// TwinCAT 3 PLC project PlcSoftware
// ProgramVersion: 3.1.4022.7
// libraries:
//   AST_V1_0, * (Deprag)
//   Tc2_MC2, * (Beckhoff Automation GmbH)
//   Tc2_MC2_Drive, * (Beckhoff Automation GmbH)
//   Tc2_Standard, * (Beckhoff Automation GmbH)
//   Tc2_System, * (Beckhoff Automation GmbH)
//   Tc2_Utilities, * (Beckhoff Automation GmbH)
//   Tc3_Module, * (Beckhoff Automation GmbH)
//   Tc3_PLCopen_OpcUa, * (Beckhoff Automation GmbH)
// project tree:
//   DUTs/ENUMs/ teAxisNames.TcDUT, teDriveState.TcDUT, teOperationMode.TcDUT, teScrewFeeders.TcDUT
//   DUTs/STRUCTs/ tsASTData.TcDUT, tsAxisPositionPoint.TcDUT, tsAxisPositions.TcDUT (not stored), tsControls.TcDUT, tsCoordinate.TcDUT, tsCoordinateBool.TcDUT (not stored), tsDriveOutputs.TcDUT, tsDriveParameter.TcDUT, tsRecipe.TcDUT (not stored), tsRecipeRow.TcDUT (not stored)
//   FBs/DRIVEs/AXIS/ FB_PTP_AXIS_ABS_CONTROL.TcPOU
//   FBs/DRIVEs/PNEU/ PNEU_DRIVE.TcPOU
//   FBs/RECIPEs/CONVERTERs/ ConvertCommandToString.TcPOU, CovertStringToCommand.TcPOU
//   FBs/RECIPEs/FILEs/ CreateRecipeFile.TcPOU, ReadRecipeFromFile.TcPOU, WriteRepcieToFile.TcPOU
//   FBs/SUBFUNCTIONs/ BLOW_DOW_SEQ.TcPOU, END_RUN_SEQ.TcPOU, HOME_RUN_SEQ.TcPOU, PICKUP_SCREW_SEQ.TcPOU, SELECT_ACTIVE_FEEDER_SEQ.TcPOU
//   GVLs/ AST40_GLV.TcGVL, CTRL_GVL.TcGVL, HMI_GLV.TcGVL, IN_OUT_GLV.TcGVL, PERSIST_GLV.TcGVL, SAFETY_IN_GLV.TcGVL, SAFETY_OUT_GLV.TcGVL
//   POUs/JIG POUs/JIG TYPE POUs/ JIG_EMPTY.TcPOU, JIG_GRAB.TcPOU, JIG_PARTPRESENT.TcPOU, JIG_TAKER.TcPOU
//   POUs/JIG POUs/ JIG001_VOLVOL125.TcPOU, JIG002_MANSCANIA2016.TcPOU, JIG003_NTG6.TcPOU, JIG004_BMW_RAM.TcPOU, JIG005_BMW_MGU.TcPOU
//   POUs/KERNEL POUs/ AST40_Controller.TcPOU, HMI_Controller.TcPOU, INIT_DataSet.TcPOU, MES_Controller.TcPOU, MOVMENT_Controller.TcPOU, OPERATION_Controller.TcPOU, RECIPE_Controller.TcPOU
//   POUs/KERNEL POUs/MES POUs/ LOCAL_COM_Controller.TcPOU, OPCUA_Controller.TcPOU
//   POUs/KERNEL POUs/OPERATIONs/ AUTOMATIC_POSITION_TEST.TcPOU, AUTOMATIC_SCREWING.TcPOU, AUTOMATIC_SCREW_PICKUP_TEST.TcPOU
//   POUs/KERNEL POUs/OPERATIONs/SUBOPERATIONs/ DROP_SCREW.TcPOU, END_RUN.TcPOU, HOME_RUN.TcPOU, PICKUP_SCREW.TcPOU, POSITION_RUN.TcPOU
//   POUs/MAIN POUs/ FAST.TcPOU, INDEP.TcPOU, JIG.TcPOU, MAIN.TcPOU
//   TASKs/ FastTask.TcTTO, PlcTask.TcTTO
// real-time tasks:
//   TASK PlcTask: cycle T#10ms, priority 12, ADS port 350
//   TASK FastTask: cycle T#10ms, priority 8, ADS port 351
// motion (NC):
//   TASK NC/PTP Task SAF: cycle T#2ms, priority 4, ADS port 501
//   TASK NC/PTP Task SVB: cycle T#10ms, priority 10, ADS port 511
//   AXIS X Axis (id 5)
//     OtherSettings: AllowMotionCmdToSlave=true
//     encoder EncType=1
//     drive DrvType=5
//       Analog: ScaleFactorActTorque=0.1
//       TimeComp: TaskDelayCycles=1
//     controller CtrType=1
//       CtrPara: PriorControlFactor=1
//         Observer: BandWidth=20
//   AXIS Y Axis (id 6)
//     OtherSettings: AllowMotionCmdToSlave=true
//     encoder EncType=1
//     drive DrvType=5
//       Analog: ScaleFactorActTorque=0.1
//       TimeComp: TaskDelayCycles=1
//     controller CtrType=1
//       CtrPara: PriorControlFactor=1
//         Observer: BandWidth=20
//   AXIS Z Axis (id 7)
//     OtherSettings: AllowMotionCmdToSlave=true
//     encoder EncType=1
//     drive DrvType=5
//       Analog: ScaleFactorActTorque=0.1
//       TimeComp: TaskDelayCycles=1
//     controller CtrType=1
//       CtrPara: PriorControlFactor=1
//         Observer: BandWidth=20
//   AXIS C Axis (id 8)
//     OtherSettings: AllowMotionCmdToSlave=true
//     encoder EncType=1
//     drive DrvType=5
//       Analog: ScaleFactorActTorque=0.1
//       TimeComp: TaskDelayCycles=1
//     controller CtrType=1
//       CtrPara: PriorControlFactor=1
//         Observer: BandWidth=20
//   AXIS Sim X Axis (id 1)
//     OtherSettings: AllowMotionCmdToSlave=true
//     encoder EncType=1
//       SoftEndMinControl: Enable=true, Range=-40
//       SoftEndMaxControl: Enable=true, Range=640
//     drive DrvType=5
//       Analog: ScaleFactorActTorque=0.1
//       TimeComp: TaskDelayCycles=1
//     controller CtrType=1
//       CtrPara: PriorControlFactor=1
//         Observer: BandWidth=20
//   AXIS Sim Y Axis (id 2)
//     OtherSettings: AllowMotionCmdToSlave=true
//     encoder EncType=1
//       SoftEndMinControl: Enable=true, Range=-193
//       SoftEndMaxControl: Enable=true, Range=530
//     drive DrvType=5
//       Analog: ScaleFactorActTorque=0.1
//       TimeComp: TaskDelayCycles=1
//     controller CtrType=1
//       CtrPara: PriorControlFactor=1
//         Observer: BandWidth=20
//   AXIS Sim Z Axis (id 3)
//     OtherSettings: AllowMotionCmdToSlave=true
//     encoder EncType=1
//       SoftEndMinControl: Enable=true, Range=-3
//       SoftEndMaxControl: Enable=true, Range=252
//     drive DrvType=5
//       Analog: ScaleFactorActTorque=0.1
//       TimeComp: TaskDelayCycles=1
//     controller CtrType=1
//       CtrPara: PriorControlFactor=1
//         Observer: BandWidth=20
//   AXIS Sim C Axis (id 4)
//     OtherSettings: AllowMotionCmdToSlave=true
//     encoder EncType=1
//       SoftEndMinControl: Enable=true
//       SoftEndMaxControl: Enable=true
//     drive DrvType=5
//       Analog: ScaleFactorActTorque=0.1
//       TimeComp: TaskDelayCycles=1
//     controller CtrType=1
//       CtrPara: PriorControlFactor=1
//         Observer: BandWidth=20
// variable links:
//   PlcSoftware/PlcSoftware Instance <-> NC/PTP Task SAF/Axes/Sim C Axis
//     PlcTask Inputs/IN_OUT_GLV.G_aAxisReferencies[4].NcToPlc <-> Outputs/ToPlc
//     PlcTask Outputs/IN_OUT_GLV.G_aAxisReferencies[4].PlcToNc <-> Inputs/FromPlc
//   PlcSoftware/PlcSoftware Instance <-> NC/PTP Task SAF/Axes/Sim X Axis
//     PlcTask Inputs/IN_OUT_GLV.G_aAxisReferencies[1].NcToPlc <-> Outputs/ToPlc
//     PlcTask Outputs/IN_OUT_GLV.G_aAxisReferencies[1].PlcToNc <-> Inputs/FromPlc
//   PlcSoftware/PlcSoftware Instance <-> NC/PTP Task SAF/Axes/Sim Y Axis
//     PlcTask Inputs/IN_OUT_GLV.G_aAxisReferencies[2].NcToPlc <-> Outputs/ToPlc
//     PlcTask Outputs/IN_OUT_GLV.G_aAxisReferencies[2].PlcToNc <-> Inputs/FromPlc
//   PlcSoftware/PlcSoftware Instance <-> NC/PTP Task SAF/Axes/Sim Z Axis
//     PlcTask Inputs/IN_OUT_GLV.G_aAxisReferencies[3].NcToPlc <-> Outputs/ToPlc
//     PlcTask Outputs/IN_OUT_GLV.G_aAxisReferencies[3].PlcToNc <-> Inputs/FromPlc

CONFIGURATION PlcSoftware
    RESOURCE PLC ON TwinCAT3
        TASK FastTask(INTERVAL := T#10ms, PRIORITY := 8);
        TASK PlcTask(INTERVAL := T#10ms, PRIORITY := 12);
        PROGRAM FAST WITH FastTask : FAST;
        PROGRAM MAIN WITH PlcTask : MAIN;
    END_RESOURCE
END_CONFIGURATION

// ---- DUTs/ENUMs/teAxisNames.TcDUT
TYPE teAxisNames :
(
	CE_AXIS_X:=1,			// X-axis drive
	CE_AXIS_Y,				// Y-axis drive
	CE_AXIS_Z,				// Z-axis drive
	CE_AXIS_C 				// C-axis drive
);
END_TYPE

// ---- DUTs/ENUMs/teDriveState.TcDUT
TYPE teDriveState :
(
	MOVESTATE_INIT,
	MOVESTATE_ENABLE,
	MOVESTATE_AUTO,
	MOVESTATE_MANUAL,
	MOVESTATE_IDLE,
	MOVESTATE_ERROR,
	MOVESTATE_RESET
) UDINT;
END_TYPE

// ---- DUTs/ENUMs/teOperationMode.TcDUT
TYPE teOperationMode :
(
	OPMODE_REFERENCETEACH,
	OPMODE_AUTOSCREWING,
	OPMODE_PICKUPTEST,
	OPMODE_POSITIONTEST
) UDINT;
END_TYPE

// ---- DUTs/ENUMs/teScrewFeeders.TcDUT
TYPE teScrewFeeders :
(
	CE_SCREW_FEED_1:=1,
	CE_SCREW_FEED_2,
	CE_SCREW_FEED_3,
	CE_SCREW_FEED_4
);
END_TYPE

// ---- DUTs/STRUCTs/tsASTData.TcDUT
TYPE tsASTData :
STRUCT
	Start:			BOOL;
	Prog:			INT;
	DataSaved:		BOOL;
	
	OK:				BOOL;
	NOK:			BOOL;
	Ready:			BOOL;
	DataAvailable:	BOOL;
	
	Status:			INT;
	Step:			DINT;
	MinTorque:		REAL;
	MaxTorque:		REAL;
	Torque:			REAL;
	MinAngle:		DINT;
	MaxAngle:		DINT;
	Angle:			REAL;
	Started:		BOOL;
END_STRUCT
END_TYPE

// ---- DUTs/STRUCTs/tsAxisPositionPoint.TcDUT
TYPE tsAxisPositionPoint :
STRUCT
	Name			: STRING;
	Description		: STRING;
	Target			: LREAL;
END_STRUCT
END_TYPE

// ---- DUTs/STRUCTs/tsControls.TcDUT
TYPE tsControls :
STRUCT
	PowerOn:					BOOL:=TRUE;
	AutoMode:					BOOL:=0;						//Automaic/Manual mode switch
	ErrorExist:					BOOL;  							//Error exist
	ErrorACK:					BOOL;							//Error acknowledge
	ManualMoveMode:				BOOL:=TRUE;						//0:= stepper, 1:= continous
	
	OperationMode:				INT:=1;							//0:= manual, 1:= automatic seq 01 ... 

	Override:					LREAL:=100;						//Main overrride value
	ManualOverride:				LREAL:=20;						//Maximum manual override value
	StepSize:					LREAL:=0.1;						//Manual jog step size
	MaximumVelocity:			LREAL:=600;						//Maximum velocity
	
	ActualPosition:				tsCoordinate;	
	TargetPosition:				tsCoordinate;	
END_STRUCT
END_TYPE

// ---- DUTs/STRUCTs/tsCoordinate.TcDUT
TYPE tsCoordinate :
STRUCT
	X: LREAL;
	Y: LREAL;
	Z: LREAL;
	C: LREAL;
END_STRUCT
END_TYPE

// ---- DUTs/STRUCTs/tsDriveOutputs.TcDUT
TYPE tsDriveOutputs :
STRUCT
	PowerOut: 			ST_McOutputs;
	ResetOut: 				ST_McOutputs;
	MoveAbsoluteOut: 		ST_McOutputs;
	MoveJogOut:				ST_McOutputs;
	MoveHalt:				ST_McOutputs;
END_STRUCT
END_TYPE

// ---- DUTs/STRUCTs/tsDriveParameter.TcDUT
TYPE tsDriveParameter :
STRUCT
	PositionMin:		LREAL;
	PositionMax:		LREAL;
	PositionOffset:		LREAL;	
END_STRUCT
END_TYPE

// ---- GVLs/AST40_GLV.TcGVL
VAR_GLOBAL
	G_sAST40_Data:				tsASTData;					//Contains all of AST40 datas	
	
	G_fbAST40:				FB_AST40;					// FB instance of the AST40
	G_sAST40:				tAST40;						// struct contains 'control', 'state' and 'data'
	
	G_sTx					AT%I*: tAST40Rx; 			// struct for the input mapping 
	G_sRx 					AT%Q*: tAST40Tx; 			// struct for the output mapping
END_VAR

// ---- GVLs/CTRL_GVL.TcGVL
VAR_GLOBAL
	G_sControl:						tsControls;						//Control data	

	G_sAxisReady:					tsCoordinateBool;				//Axis ready to move state container
	G_sAxisDone:					tsCoordinateBool;				//Axis done state container
	G_sAckAxisDone:					tsCoordinateBool;				//Axis done acknowledge container
	
	G_sStartToPos:					tsCoordinateBool;				//Start to position
END_VAR

// ---- GVLs/HMI_GLV.TcGVL
VAR_GLOBAL
	G_sHMIAxisJogForward:				tsCoordinateBool;				//Axis jog forward
	G_sHMIAxisJogBackward:				tsCoordinateBool;				//Axis jog backward
END_VAR

// ---- GVLs/IN_OUT_GLV.TcGVL
VAR_GLOBAL
	//Axis referencies for driving
	G_aAxisReferencies:				ARRAY [1..CE_AXIS_C] OF AXIS_REF;
	
	//Input linkable definition
	I_xFeedbackES           		AT%I* :BOOL;
	I_xVacuumIntake_OK				AT%I*: BOOL;
	I_xStart						AT%I*: BOOL;
	I_xLightGridError				AT%I*: BOOL;
	I_xSafetyDoorClosed				AT%I*: BOOL;
	I_xServoFanDiag					AT%I*: BOOL;
	I_xPneumatic_OK					AT%I*: BOOL;
	I_xScrewFeed_READY			 	AT%I*: ARRAY[1..CE_SCREW_FEED_4] OF BOOL;
	I_xScrewFeeder_POS				AT%I*: ARRAY[1..CE_SCREW_FEED_4] OF BOOL;
	I_xPartSensor1					AT%I*: BOOL;
	I_xPartSensor2					AT%I*: BOOL;
	I_xEpInputBox01					AT%I*: ARRAY[1..16] OF BOOL;	
	I_xEpInputBox02					AT%I*: ARRAY[1..16] OF BOOL;
	
	//Output linkable definition
	Q_axScrewFeeders					AT%Q*:ARRAY [1..CE_SCREW_FEED_4] OF BOOL;
	Q_xValve_PressureSwitch				AT%Q*: BOOL;
	Q_xBlowValve						AT%Q*: BOOL;
	Q_xVacuumValve						AT%Q*: BOOL;
END_VAR

// ---- GVLs/PERSIST_GLV.TcGVL
VAR_GLOBAL PERSISTENT
	G_xExistCAxis:					BOOL:=TRUE;							//TRUE:=Exist C-Axis, FALSE:=Not exist C-Axis
	//Individual axis positions like fider position...
	G_asIndividualAxisPositions:		ARRAY [1..CE_AXIS_C] OF tsAxisPositions;
	//Min/Max/Offset parameters for drives...
	G_asDriveParameters:				ARRAY [1..CE_AXIS_C] OF tsDriveParameter:= [(PositionMin:=-40.00,	PositionMax:=640.00,		PositionOffset:=-293.00),	(*X-Axis initial parameters*)
																					(PositionMin:=-193.00,	PositionMax:=530.00,	PositionOffset:=240.00),		(*Y-Axis initial parameters*)
																					(PositionMin:=-3,		PositionMax:=252,		PositionOffset:=127.00), 		(*Z-Axis initial parameters*)
																					(PositionMin:=0,		PositionMax:=0,			PositionOffset:=0.00)];			(*C-Axis initial parameters*)
END_VAR

// ---- GVLs/SAFETY_IN_GLV.TcGVL
VAR_GLOBAL
	I_xTsEstopCH1					AT%I*: BOOL;
	I_xTsEstopCH2					AT%I*: BOOL;
	I_xTsE_Stop			 			AT%I*: BOOL;
	I_xTsCommErr					AT%I*: BOOL;
	I_xTsLightGridOK				AT%I*: BOOL;
	I_xTsFBErr						AT%I*: BOOL;
END_VAR

// ---- GVLs/SAFETY_OUT_GLV.TcGVL
VAR_GLOBAL
	Q_xTsFB_E_Stop					AT%Q*: BOOL;
	Q_xTsEStopReset                 AT%Q*: BOOL;
	Q_xTsTwinsafeRun				AT%Q*: BOOL;
	Q_xTsErrAck						AT%Q*: BOOL;
END_VAR

// ---- POUs/MAIN POUs/FAST.TcPOU
PROGRAM FAST
VAR
	tpEStopAck:		TP;
	rtErrorACK: 	R_TRIG;
END_VAR


Q_xTsTwinsafeRun := NOT I_xTsCommErr;
Q_xTsErrAck := I_xTsCommErr;

rtErrorAck(CLK:= G_sControl.ErrorAck, Q=> G_sControl.ErrorAck);
tpEStopAck(IN:= rtErrorAck.Q, pt:= T#100MS);

Q_xTsFB_E_Stop :=I_xFeedbackES;
Q_xTsEstopReset := (tpEStopAck.ET > T#100MS AND tpEStopAck.ET < T#300MS);

END_PROGRAM

// ---- POUs/MAIN POUs/MAIN.TcPOU
PROGRAM MAIN
VAR
	bInit:					BOOL:=TRUE;	
	xOpenVisu:				BOOL;
	sMachineName:			STRING;
	sVisuURL:				STRING;
	fbStartProcess:			NT_StartProcess;
	fbGetHostName:			FB_GetHostName;
END_VAR

(*
fbGetHostName(	 
				 bExecute:= TRUE,
				 sHostName=>sMachineName);
sVisuURL:= CONCAT('--app=https://huszwsap10:1020/Default.html?TargetHost=', sMachineName);
fbStartProcess(
				 NETID:= '',
				 PATHSTR:= 'C:\Program Files (x86)\Google\Chrome\Application\chrome.exe',
				 DIRNAME:= 'C:\Program Files (x86)\Google\Chrome\Application',
				 COMNDLINE:= sVisuURL,
				 START:= (LEN (sMachineName)>0),
				 TMOUT:= T#20S);
*)		
		 
INIT_DataSet();
//RECIPE_Controller();
//DRIVE_Controller();
MOVMENT_Controller();
OPERATION_Controller();
HMI_Controller();

END_PROGRAM

// ---- POUs/KERNEL POUs/INIT_DataSet.TcPOU
PROGRAM INIT_DataSet
VAR
	xWriteExecute:					BOOL;
	xErrorInProces:					BOOL:=FALSE;
	xCounter:						INT:=1;
	
	fbMC_WriteOffsetParameterX: 		MC_WriteParameter;
	fbMC_WriteMinParameterX: 		MC_WriteParameter;
	fbMC_WriteMaxParameterX: 		MC_WriteParameter;
	
	fbMC_WriteOffsetParameterY: 		MC_WriteParameter;
	fbMC_WriteMinParameterY: 		MC_WriteParameter;
	fbMC_WriteMaxParameterY: 		MC_WriteParameter;
	
	fbMC_WriteOffsetParameterZ: 		MC_WriteParameter;
	fbMC_WriteMinParameterZ: 		MC_WriteParameter;
	fbMC_WriteMaxParameterZ: 		MC_WriteParameter;
	
	fbMC_WriteOffsetParameterC: 		MC_WriteParameter;
	fbMC_WriteMinParameterC: 		MC_WriteParameter;
	fbMC_WriteMaxParameterC: 		MC_WriteParameter;
END_VAR

//X-Axis Write parameter
fbMC_WriteOffsetParameterX(
					Axis:= G_aAxisReferencies[CE_AXIS_X], 
					Execute:= xWriteExecute, 
					ParameterNumber:= 1042, 
					Value:= G_asDriveParameters[CE_AXIS_X].PositionOffset,
					Error=>  xErrorInProces
					);
fbMC_WriteMinParameterX(
					Axis:= G_aAxisReferencies[CE_AXIS_X], 
					Execute:= xWriteExecute, 
					ParameterNumber:= 3, 
					Value:= G_asDriveParameters[CE_AXIS_X].PositionMin,
					Error=>  xErrorInProces
					);
fbMC_WriteMaxParameterX(
					Axis:= G_aAxisReferencies[CE_AXIS_X], 
					Execute:= xWriteExecute, 
					ParameterNumber:= 2, 
					Value:= G_asDriveParameters[CE_AXIS_X].PositionMax,
					Error=>  xErrorInProces
					);
//Y-Axis Write paramater
fbMC_WriteOffsetParameterY(
					Axis:= G_aAxisReferencies[CE_AXIS_Y], 
					Execute:= xWriteExecute, 
					ParameterNumber:= 1042, 
					Value:= G_asDriveParameters[CE_AXIS_Y].PositionOffset,
					Error=>  xErrorInProces
					);
fbMC_WriteMinParameterY(
					Axis:= G_aAxisReferencies[CE_AXIS_Y], 
					Execute:= xWriteExecute, 
					ParameterNumber:= 3, 
					Value:= G_asDriveParameters[CE_AXIS_Y].PositionMin,
					Error=>  xErrorInProces
					);
fbMC_WriteMaxParameterY(
					Axis:= G_aAxisReferencies[CE_AXIS_Y], 
					Execute:= xWriteExecute, 
					ParameterNumber:= 2, 
					Value:= G_asDriveParameters[CE_AXIS_Y].PositionMax,
					Error=>  xErrorInProces
					);
//Z-Axis Write parameter
fbMC_WriteOffsetParameterZ(
					Axis:= G_aAxisReferencies[CE_AXIS_Z], 
					Execute:= xWriteExecute, 
					ParameterNumber:= 1042, 
					Value:= G_asDriveParameters[CE_AXIS_Z].PositionOffset,
					Error=>  xErrorInProces
					);
fbMC_WriteMinParameterZ(
					Axis:= G_aAxisReferencies[CE_AXIS_Z], 
					Execute:= xWriteExecute, 
					ParameterNumber:= 3, 
					Value:= G_asDriveParameters[CE_AXIS_Z].PositionMin,
					Error=>  xErrorInProces
					);
fbMC_WriteMaxParameterZ(
					Axis:= G_aAxisReferencies[CE_AXIS_Z], 
					Execute:= xWriteExecute, 
					ParameterNumber:= 2, 
					Value:= G_asDriveParameters[CE_AXIS_Z].PositionMax,
					Error=>  xErrorInProces
					);
//C-Axis Write parameter
fbMC_WriteOffsetParameterC(
					Axis:= G_aAxisReferencies[CE_AXIS_C], 
					Execute:= xWriteExecute, 
					ParameterNumber:= 1042, 
					Value:= G_asDriveParameters[CE_AXIS_C].PositionOffset,
					Error=>  xErrorInProces
					);
fbMC_WriteMinParameterC(
					Axis:= G_aAxisReferencies[CE_AXIS_C], 
					Execute:= xWriteExecute, 
					ParameterNumber:= 3, 
					Value:= G_asDriveParameters[CE_AXIS_C].PositionMin,
					Error=>  xErrorInProces
					);
fbMC_WriteMaxParameterC(
					Axis:= G_aAxisReferencies[CE_AXIS_C], 
					Execute:= xWriteExecute, 
					ParameterNumber:= 2, 
					Value:= G_asDriveParameters[CE_AXIS_C].PositionMax,
					Error=>  xErrorInProces
					);
					
IF xErrorInProces THEN
	xWriteExecute:= FALSE;
ELSE
	xWriteExecute:= TRUE;
END_IF

END_PROGRAM

// ---- POUs/KERNEL POUs/MOVMENT_Controller.TcPOU
PROGRAM MOVMENT_Controller
VAR
	X_Axis:				FB_PTP_AXIS_ABS_CONTROL;
	Y_Axis:				FB_PTP_AXIS_ABS_CONTROL;
	Z_Axis:				FB_PTP_AXIS_ABS_CONTROL;
	
	eJogMode: 				E_JogMode;
END_VAR

IF (G_sControl.ManualMoveMode) THEN
	eJogMode:= MC_JOGMODE_CONTINOUS;
ELSE
	eJogMode:= MC_JOGMODE_INCHING;
END_IF

ACT_AXIS_CTRL();

ACTION ACT_AXIS_CTRL:
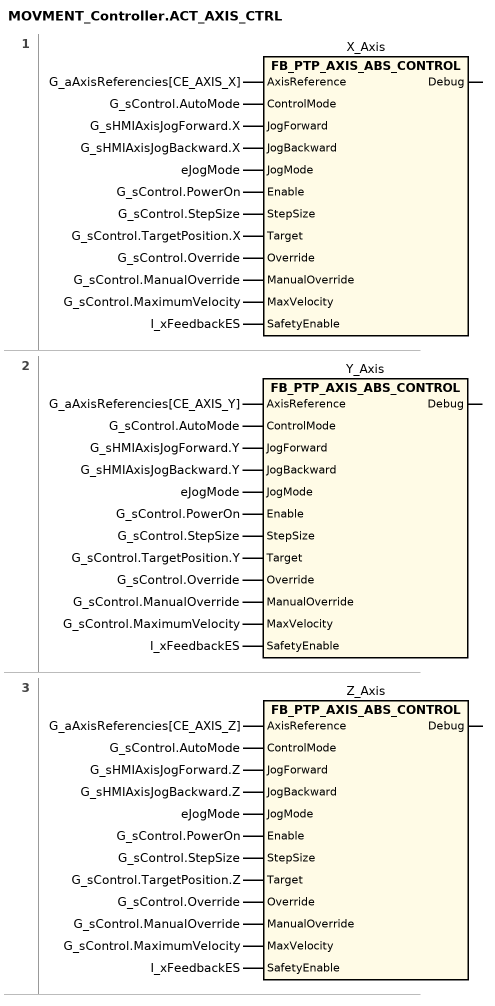
// NETWORK 1
X_Axis(
    AxisReference := G_aAxisReferencies[CE_AXIS_X],
    ControlMode := G_sControl.AutoMode,
    JogForward := G_sHMIAxisJogForward.X,
    JogBackward := G_sHMIAxisJogBackward.X,
    JogMode := eJogMode,
    Enable := G_sControl.PowerOn,
    StepSize := G_sControl.StepSize,
    Target := G_sControl.TargetPosition.X,
    Override := G_sControl.Override,
    ManualOverride := G_sControl.ManualOverride,
    MaxVelocity := G_sControl.MaximumVelocity,
    SafetyEnable := I_xFeedbackES); // FB_PTP_AXIS_ABS_CONTROL

// NETWORK 2
Y_Axis(
    AxisReference := G_aAxisReferencies[CE_AXIS_Y],
    ControlMode := G_sControl.AutoMode,
    JogForward := G_sHMIAxisJogForward.Y,
    JogBackward := G_sHMIAxisJogBackward.Y,
    JogMode := eJogMode,
    Enable := G_sControl.PowerOn,
    StepSize := G_sControl.StepSize,
    Target := G_sControl.TargetPosition.Y,
    Override := G_sControl.Override,
    ManualOverride := G_sControl.ManualOverride,
    MaxVelocity := G_sControl.MaximumVelocity,
    SafetyEnable := I_xFeedbackES); // FB_PTP_AXIS_ABS_CONTROL

// NETWORK 3
Z_Axis(
    AxisReference := G_aAxisReferencies[CE_AXIS_Z],
    ControlMode := G_sControl.AutoMode,
    JogForward := G_sHMIAxisJogForward.Z,
    JogBackward := G_sHMIAxisJogBackward.Z,
    JogMode := eJogMode,
    Enable := G_sControl.PowerOn,
    StepSize := G_sControl.StepSize,
    Target := G_sControl.TargetPosition.Z,
    Override := G_sControl.Override,
    ManualOverride := G_sControl.ManualOverride,
    MaxVelocity := G_sControl.MaximumVelocity,
    SafetyEnable := I_xFeedbackES); // FB_PTP_AXIS_ABS_CONTROL
END_ACTION

END_PROGRAM

// ---- FBs/DRIVEs/AXIS/FB_PTP_AXIS_ABS_CONTROL.TcPOU
FUNCTION_BLOCK FB_PTP_AXIS_ABS_CONTROL
VAR_INPUT
	ControlMode:				BOOL;					// Manual (JOG mode) or Automatic (ABSOLUTE PTP mode) | 0:=Manual 1:=Automatic
	
	JogForward:					BOOL;					// Jog the axis in forward direction (based on the JogMode)
	JogBackward:				BOOL;					// Jog the axis in forward direction (based on the JogMode)
	JogMode:					E_JogMode;				// Selected Jog mode is determin the manual movement method stepper or continous
	
	Enable:						BOOL;					// Enable axis
	Start:						BOOL;					// Start to position in automatic mode
	StepSize:					LREAL;					// Stepsize (like: 0.1mm, 0.2mm, 0.5mm, 1mm ....)
	Target:						LREAL;					// Target position in automatic mode
	Override:					LREAL;					// Overall axis override (0-100%)
	ManualOverride:				LREAL;					// Manual override (0-20%)
	MaxVelocity:				LREAL;					// Maximum axis velocity (0-600)
	
	SafetyEnable:				BOOL;
END_VAR
VAR_IN_OUT
	AxisReference:				AXIS_REF;				// Contains all referencies for the NC Axis
END_VAR
VAR_OUTPUT
	Debug:						tsDriveOutputs;			// Debug function block output struct
END_VAR
VAR
	AxisState:					teDriveState;			// Contains the control actual state.
	
	LastTarget:					LREAL;
	
	MoveAbs:					MC_MoveAbsolute;		
	MoveJog:					MC_Jog;
	MoveHalt:					MC_Halt;
	Reset:						MC_Reset;
	SoEReset:					FB_SoEReset;
	Power:						MC_Power;
END_VAR

(* update the axis status at the beginning of each cycle *)
AxisReference();

(* axis drive state machine *)
CASE AxisState OF
	
	MOVESTATE_INIT:																		(* initialisation *)
		MoveAbs.Execute :=			FALSE;
		Reset.Execute :=			FALSE;
		AxisState := 				MOVESTATE_ENABLE;
		
		IF NOT SafetyEnable THEN 
			AxisState := MOVESTATE_ERROR;
		END_IF
	
	MOVESTATE_ENABLE:																	(* enabel power *)
		Power.Enable :=				TRUE;
		Power.BufferMode :=			MC_Aborting;
		
		IF Power.Status THEN
			AxisState := MOVESTATE_IDLE;
		ELSIF Power.Error THEN
			Power.Enable :=				FALSE;
			AxisState := MOVESTATE_ERROR;
		END_IF
	
	MOVESTATE_IDLE:																		(* Idle state stay here until the next command *)			
		IF ControlMode AND Start AND SafetyEnable THEN
			AxisState := MOVESTATE_AUTO;
			
		ELSIF NOT ControlMode AND (JogForward OR JogBackward) AND SafetyEnable THEN
			AxisState := MOVESTATE_MANUAL;
			
		ELSIF NOT SafetyEnable THEN 
			Power.Enable :=				FALSE;
			AxisState := MOVESTATE_ERROR;
		
		END_IF
		
	MOVESTATE_AUTO:																		(* automatic movment mode *)
		IF LastTarget=target AND NOT Start THEN
			AxisState := MOVESTATE_IDLE;
		ELSE
			MoveAbs.Position := 	target;
			MoveAbs.Velocity := 	MaxVelocity;
			MoveAbs.BufferMode := 	MC_Aborting;
			MoveAbs.Execute := 		TRUE;
			
			IF MoveAbs.Done AND NOT Start THEN
				MoveAbs.Execute := FALSE;
				AxisState := MOVESTATE_IDLE;
				
			ELSIF MoveAbs.CommandAborted OR MoveAbs.Error THEN
				AxisState := MOVESTATE_ERROR;
			END_IF	
		END_IF
	
	MOVESTATE_MANUAL:																	(* manual movement mode *)
		MoveJog.Position := 	StepSize;
		MoveJog.Mode := 		JogMode;
		MoveJog.Velocity := 	(ManualOverride*MaxVelocity)/100;						(* speed reduction in manual movement mode *)
		
		IF MoveJog.Done AND NOT MoveHalt.Done THEN
			MoveHalt.Execute := 	TRUE;
			MoveHalt.BufferMode := 	MC_Aborting;
			
		ELSIF MoveHalt.Done AND NOT MoveJog.Done THEN
				MoveHalt.Execute := FALSE;
				AxisState := MOVESTATE_IDLE;

		ELSIF MoveJog.CommandAborted OR MoveAbs.Error OR MoveHalt.CommandAborted THEN
				AxisState := MOVESTATE_ERROR;	
		END_IF
	
	MOVESTATE_ERROR:																	(* in error state *)
		IF AxisReference.Status.Error THEN
			AxisState := MOVESTATE_RESET;												(* axis error requires reset *)
			
		ELSE
			AxisState := MOVESTATE_INIT;												(* function block errors don't need a reset *)
			
		END_IF
	
	MOVESTATE_RESET:																	(* reset axis functions *)
		Power.Enable :=				FALSE;		
		SoEReset.Execute := TRUE;
		SoEReset.Timeout := T#10S;
		IF NOT SoEReset.Busy THEN
			SoEReset.Execute := FALSE;
			Reset.Execute := TRUE;
			IF Reset.Done THEN
				AxisState := MOVESTATE_INIT;	
			ELSIF Reset.Error THEN
				AxisState := MOVESTATE_INIT; 												(* can't do anything here *)
			END_IF
		END_IF
	
END_CASE

ACT_MOVE();
ACT_POWER();
ACT_RESET();

ACTION ACT_MOVE:
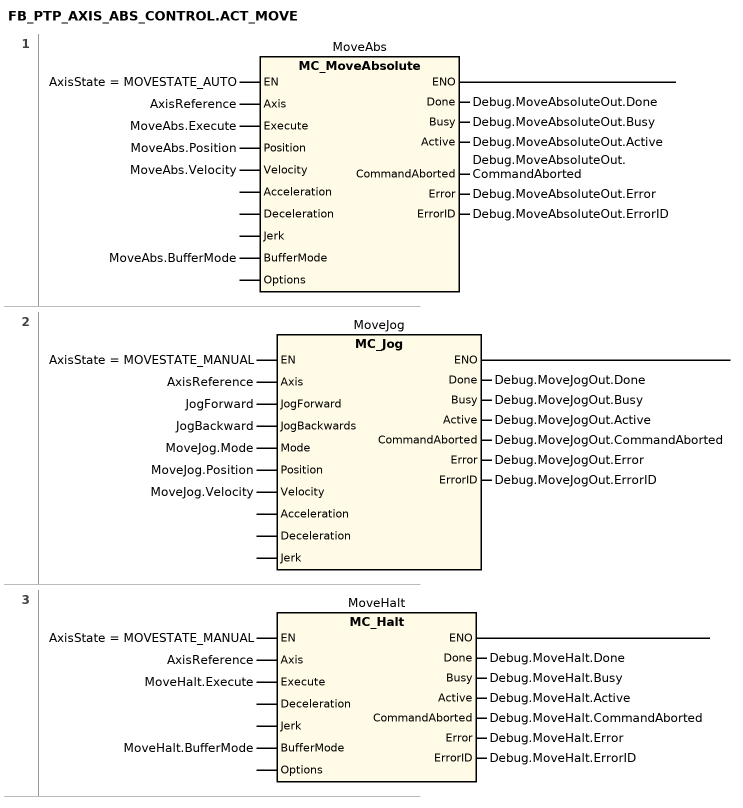
// NETWORK 1
IF AxisState = MOVESTATE_AUTO THEN
    MoveAbs(
        Axis := AxisReference,
        Execute := MoveAbs.Execute,
        Position := MoveAbs.Position,
        Velocity := MoveAbs.Velocity,
        BufferMode := MoveAbs.BufferMode,
        Done => Debug.MoveAbsoluteOut.Done,
        Busy => Debug.MoveAbsoluteOut.Busy,
        Active => Debug.MoveAbsoluteOut.Active,
        CommandAborted => Debug.MoveAbsoluteOut.CommandAborted,
        Error => Debug.MoveAbsoluteOut.Error,
        ErrorID => Debug.MoveAbsoluteOut.ErrorID); // MC_MoveAbsolute
END_IF

// NETWORK 2
IF AxisState = MOVESTATE_MANUAL THEN
    MoveJog(
        Axis := AxisReference,
        JogForward := JogForward,
        JogBackwards := JogBackward,
        Mode := MoveJog.Mode,
        Position := MoveJog.Position,
        Velocity := MoveJog.Velocity,
        Done => Debug.MoveJogOut.Done,
        Busy => Debug.MoveJogOut.Busy,
        Active => Debug.MoveJogOut.Active,
        CommandAborted => Debug.MoveJogOut.CommandAborted,
        Error => Debug.MoveJogOut.Error,
        ErrorID => Debug.MoveJogOut.ErrorID); // MC_Jog
END_IF

// NETWORK 3
IF AxisState = MOVESTATE_MANUAL THEN
    MoveHalt(
        Axis := AxisReference,
        Execute := MoveHalt.Execute,
        BufferMode := MoveHalt.BufferMode,
        Done => Debug.MoveHalt.Done,
        Busy => Debug.MoveHalt.Busy,
        Active => Debug.MoveHalt.Active,
        CommandAborted => Debug.MoveHalt.CommandAborted,
        Error => Debug.MoveHalt.Error,
        ErrorID => Debug.MoveHalt.ErrorID); // MC_Halt
END_IF
END_ACTION

ACTION ACT_POWER:
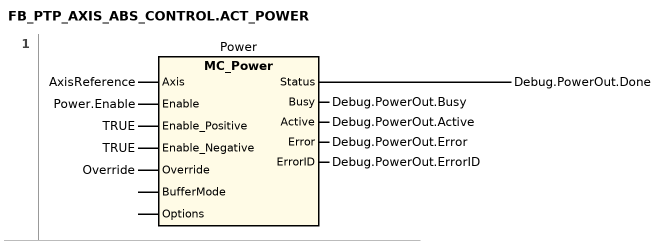
// NETWORK 1
Power(
    Axis := AxisReference,
    Enable := Power.Enable,
    Enable_Positive := TRUE,
    Enable_Negative := TRUE,
    Override := Override,
    Busy => Debug.PowerOut.Busy,
    Active => Debug.PowerOut.Active,
    Error => Debug.PowerOut.Error,
    ErrorID => Debug.PowerOut.ErrorID); // MC_Power
Debug.PowerOut.Done := Power.Status;
END_ACTION

ACTION ACT_RESET:
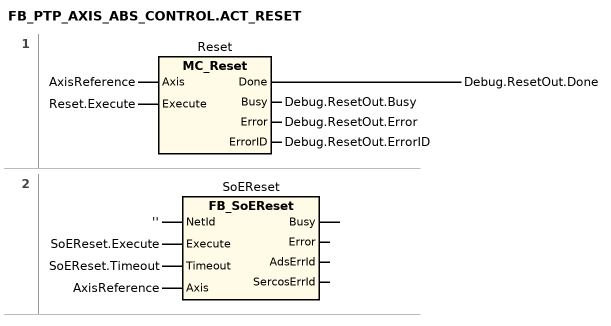
// NETWORK 1
Reset(
    Axis := AxisReference,
    Execute := Reset.Execute,
    Busy => Debug.ResetOut.Busy,
    Error => Debug.ResetOut.Error,
    ErrorID => Debug.ResetOut.ErrorID); // MC_Reset
Debug.ResetOut.Done := Reset.Done;

// NETWORK 2
SoEReset(NetId := '', Execute := SoEReset.Execute, Timeout := SoEReset.Timeout, Axis := AxisReference); // FB_SoEReset
END_ACTION

END_FUNCTION_BLOCK

// ---- POUs/KERNEL POUs/OPERATION_Controller.TcPOU
PROGRAM OPERATION_Controller
VAR	
	xHomeRunExecute:		BOOL;
	xDone:					BOOL;
	xHomeOK:				BOOL;
	
	rtControlOn:			R_TRIG;
	rtHomeRunDone:			R_TRIG;
	
	fbHOME_RUN:				HOME_RUN_SEQ;
END_VAR

rtControlOn(CLK:=G_sControl.AutoMode);
rtHomeRunDone(CLK:=xDone);

IF rtControlOn.Q AND G_sControl.PowerOn AND (NOT G_sControl.ErrorExist) THEN 
	xHomeRunExecute:=TRUE; 
END_IF

IF rtHomeRunDone.Q THEN 
	xHomeOK:=TRUE; 
END_IF

fbHOME_RUN(	xExecute:=xHomeRunExecute, xDone:=xDone);

END_PROGRAM

// ---- FBs/SUBFUNCTIONs/HOME_RUN_SEQ.TcPOU
FUNCTION_BLOCK HOME_RUN_SEQ
VAR_IN_OUT
	xExecute:		BOOL;
	xDone:			BOOL;
END_VAR
VAR_OUTPUT
	
END_VAR
VAR
	tpReset:			TP;
	rtDone:				R_TRIG;
	rtExecute:			R_TRIG;
	ftTimePulse:		F_TRIG;
	tpTimePulse:		TP;
	fbBLOW_DOW_SEQ: 	BLOW_DOW_SEQ;
	xBlowDownExecute:	BOOL;
	fbEND_RUN_SEQ:		END_RUN_SEQ;
	xEndRunExecute:		BOOL;
	
	lrTargetPos:		LREAL;
	xTransCondition:	BOOL;	
	xTransRelease:		BOOL;
	SFCInit:			BOOL;
	SFCReset:			BOOL;	
	SFCError:			BOOL;
	
END_VAR

rtDone(CLK:=xDone);
IF rtDone.Q THEN
	xTransRelease:=FALSE;	
	SFCReset:=TRUE;
	xExecute:=FALSE;
END_IF
rtExecute(CLK:=xExecute);
IF rtExecute.Q THEN
	xTransRelease:=TRUE;
END_IF

aSEQ_ACT();

tpReset(IN:=SFCError, PT:=T#250MS);
SFCReset:= tpReset.Q;

ACTION ACK_DONE_AXIS_active:
IF G_sAxisDone.X OR G_sAxisDone.Y OR G_sAxisDone.Z OR G_sAxisDone.c THEN
	G_sAckAxisDone.X:=TRUE;
	G_sAckAxisDone.Y:=TRUE;
	G_sAckAxisDone.Z:=TRUE;
	G_sAckAxisDone.C:=TRUE;
ELSE
	G_sAckAxisDone.X:=FALSE;
	G_sAckAxisDone.Y:=FALSE;
	G_sAckAxisDone.Z:=FALSE;
	G_sAckAxisDone.C:=FALSE;
END_IF

xTransCondition:= NOT G_sAckAxisDone.X AND NOT G_sAckAxisDone.Y AND NOT G_sAckAxisDone.Z AND NOT G_sAckAxisDone.C;
END_ACTION

ACTION aSEQ_ACT:
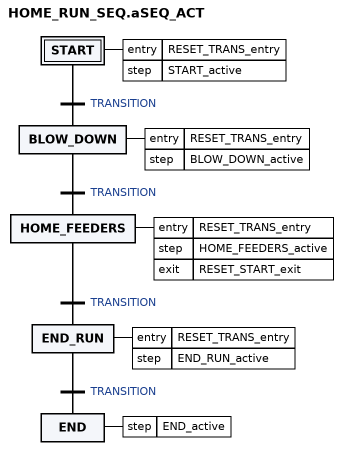
INITIAL_STEP START:
    RESET_TRANS_entry(P1);  // entry action
    START_active(N);  // step action
END_STEP
TRANSITION FROM START TO BLOW_DOWN
    := TRANSITION;
END_TRANSITION
STEP BLOW_DOWN:
    RESET_TRANS_entry(P1);  // entry action
    BLOW_DOWN_active(N);  // step action
END_STEP
TRANSITION FROM BLOW_DOWN TO HOME_FEEDERS
    := TRANSITION;
END_TRANSITION
STEP HOME_FEEDERS:
    RESET_TRANS_entry(P1);  // entry action
    HOME_FEEDERS_active(N);  // step action
    RESET_START_exit(P0);  // exit action
END_STEP
TRANSITION FROM HOME_FEEDERS TO END_RUN
    := TRANSITION;
END_TRANSITION
STEP END_RUN:
    RESET_TRANS_entry(P1);  // entry action
    END_RUN_active(N);  // step action
END_STEP
TRANSITION FROM END_RUN TO END
    := TRANSITION;
END_TRANSITION
STEP END:
    END_active(N);  // step action
END_STEP
END_ACTION

ACTION BLOW_DOWN_active:
xBlowDownExecute:=TRUE;
fbBLOW_DOW_SEQ(	xExecute:=xBlowDownExecute, xDone:=xTransCondition);
END_ACTION

ACTION END_active:
xDone:=TRUE;
xTransCondition:=FALSE;
END_ACTION

ACTION END_RUN_active:
xEndRunExecute:=TRUE;
fbEND_RUN_SEQ(xExecute:=xEndRunExecute,xJigEndDone:=TRUE, xDone:=xTransCondition);
END_ACTION

ACTION HOME_FEEDERS_active:
xTransCondition:=true;
END_ACTION

ACTION RESET_START_exit:
IF G_sAxisDone.X OR G_sAxisDone.Y OR G_sAxisDone.Z OR G_sAxisDone.c THEN
	G_sAckAxisDone.X:=TRUE;
	G_sAckAxisDone.Y:=TRUE;
	G_sAckAxisDone.Z:=TRUE;
	G_sAckAxisDone.C:=TRUE;
ELSE
	G_sAckAxisDone.X:=FALSE;
	G_sAckAxisDone.Y:=FALSE;
	G_sAckAxisDone.Z:=FALSE;
	G_sAckAxisDone.C:=FALSE;
	
	G_sStartToPos.X:=FALSE;
	G_sStartToPos.Y:=FALSE;
	G_sStartToPos.Z:=FALSE;
	G_sStartToPos.C:=FALSE;
END_IF
END_ACTION

ACTION RESET_TRANS_entry:
xTransCondition:= false;
END_ACTION

ACTION START_active:
xDone:=FALSE;
xTransCondition:= NOT xDone;
END_ACTION

TRANSITION TRANSITION:
xTransRelease AND xTransCondition
END_TRANSITION

END_FUNCTION_BLOCK

// ---- FBs/SUBFUNCTIONs/BLOW_DOW_SEQ.TcPOU
FUNCTION_BLOCK BLOW_DOW_SEQ
VAR_IN_OUT
	xExecute:		BOOL;
	xDone:			BOOL;
END_VAR
VAR_OUTPUT
	
END_VAR
VAR
	tpReset:			TP;
	rtDone:				R_TRIG;
	rtExecute:			R_TRIG;
	ftTimePulse:		F_TRIG;
	tpTimePulse:		TP;
	lrTargetPos:		LREAL;
	xTransCondition:	BOOL;	
	xTransRelease:		BOOL;
	SFCInit:			BOOL;
	SFCReset:			BOOL;	
	SFCError:			BOOL;
END_VAR

rtDone(CLK:=xDone);
IF rtDone.Q THEN
	xTransRelease:=FALSE;	
	SFCReset:=TRUE;
	xExecute:=FALSE;
END_IF

rtExecute(CLK:=xExecute);
IF rtExecute.Q THEN
	xTransRelease:=TRUE;
END_IF

aSEQ_ACT();

tpReset(IN:=SFCError, PT:=T#250MS);
SFCReset:= tpReset.Q;

ACTION ACK_DONE_AXIS_active:
IF G_sAxisDone.X OR G_sAxisDone.Y OR G_sAxisDone.Z OR G_sAxisDone.c THEN
	G_sAckAxisDone.X:=TRUE;
	G_sAckAxisDone.Y:=TRUE;
	G_sAckAxisDone.Z:=TRUE;
	G_sAckAxisDone.C:=TRUE;
ELSE
	G_sAckAxisDone.X:=FALSE;
	G_sAckAxisDone.Y:=FALSE;
	G_sAckAxisDone.Z:=FALSE;
	G_sAckAxisDone.C:=FALSE;
END_IF

xTransCondition:= NOT G_sAckAxisDone.X AND NOT G_sAckAxisDone.Y AND NOT G_sAckAxisDone.Z AND NOT G_sAckAxisDone.C;
END_ACTION

ACTION aSEQ_ACT:
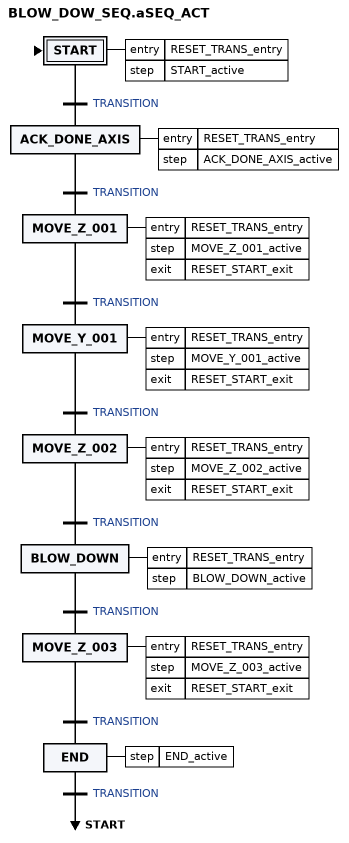
INITIAL_STEP START:
    RESET_TRANS_entry(P1);  // entry action
    START_active(N);  // step action
END_STEP
TRANSITION FROM START TO ACK_DONE_AXIS
    := TRANSITION;
END_TRANSITION
STEP ACK_DONE_AXIS:
    RESET_TRANS_entry(P1);  // entry action
    ACK_DONE_AXIS_active(N);  // step action
END_STEP
TRANSITION FROM ACK_DONE_AXIS TO MOVE_Z_001
    := TRANSITION;
END_TRANSITION
STEP MOVE_Z_001:
    RESET_TRANS_entry(P1);  // entry action
    MOVE_Z_001_active(N);  // step action
    RESET_START_exit(P0);  // exit action
END_STEP
TRANSITION FROM MOVE_Z_001 TO MOVE_Y_001
    := TRANSITION;
END_TRANSITION
STEP MOVE_Y_001:
    RESET_TRANS_entry(P1);  // entry action
    MOVE_Y_001_active(N);  // step action
    RESET_START_exit(P0);  // exit action
END_STEP
TRANSITION FROM MOVE_Y_001 TO MOVE_Z_002
    := TRANSITION;
END_TRANSITION
STEP MOVE_Z_002:
    RESET_TRANS_entry(P1);  // entry action
    MOVE_Z_002_active(N);  // step action
    RESET_START_exit(P0);  // exit action
END_STEP
TRANSITION FROM MOVE_Z_002 TO BLOW_DOWN
    := TRANSITION;
END_TRANSITION
STEP BLOW_DOWN:
    RESET_TRANS_entry(P1);  // entry action
    BLOW_DOWN_active(N);  // step action
END_STEP
TRANSITION FROM BLOW_DOWN TO MOVE_Z_003
    := TRANSITION;
END_TRANSITION
STEP MOVE_Z_003:
    RESET_TRANS_entry(P1);  // entry action
    MOVE_Z_003_active(N);  // step action
    RESET_START_exit(P0);  // exit action
END_STEP
TRANSITION FROM MOVE_Z_003 TO END
    := TRANSITION;
END_TRANSITION
STEP END:
    END_active(N);  // step action
END_STEP
TRANSITION FROM END TO START
    := TRANSITION;
END_TRANSITION
END_ACTION

ACTION BLOW_DOWN_active:
tpTimePulse(IN:=NOT tpTimePulse.Q, PT:=T#500MS);
ftTimePulse(CLK:=tpTimePulse.Q);
xTransCondition:= ftTimePulse.Q;
END_ACTION

ACTION END_active:
xDone:=TRUE;
xTransCondition:=xDone;
END_ACTION

ACTION MOVE_Y_001_active:
G_sControl.TargetPosition.Y:= G_asIndividualAxisPositions[CE_AXIS_Y].Positions[1].Target;
G_sStartToPos.Y:= TRUE;

xTransCondition:= G_sAxisDone.Y;
END_ACTION

ACTION MOVE_Z_001_active:
G_sControl.TargetPosition.Z:= G_asIndividualAxisPositions[CE_AXIS_Z].Positions[1].Target;
G_sStartToPos.Z:= TRUE;

xTransCondition:= G_sAxisDone.Z;
END_ACTION

ACTION MOVE_Z_002_active:
G_sControl.TargetPosition.Z:= G_asIndividualAxisPositions[CE_AXIS_Z].Positions[2].Target;
G_sStartToPos.Z:= TRUE;

xTransCondition:= G_sAxisDone.Z;
END_ACTION

ACTION MOVE_Z_003_active:
G_sControl.TargetPosition.Z:= G_asIndividualAxisPositions[CE_AXIS_Z].Positions[1].Target;
G_sStartToPos.Z:= TRUE;

xTransCondition:= G_sAxisDone.Z;
END_ACTION

ACTION RESET_START_exit:
IF G_sAxisDone.X OR G_sAxisDone.Y OR G_sAxisDone.Z OR G_sAxisDone.c THEN
	G_sAckAxisDone.X:=TRUE;
	G_sAckAxisDone.Y:=TRUE;
	G_sAckAxisDone.Z:=TRUE;
	G_sAckAxisDone.C:=TRUE;
ELSE
	G_sAckAxisDone.X:=FALSE;
	G_sAckAxisDone.Y:=FALSE;
	G_sAckAxisDone.Z:=FALSE;
	G_sAckAxisDone.C:=FALSE;
	
	G_sStartToPos.X:=FALSE;
	G_sStartToPos.Y:=FALSE;
	G_sStartToPos.Z:=FALSE;
	G_sStartToPos.C:=FALSE;
END_IF
END_ACTION

ACTION RESET_TRANS_entry:
xTransCondition:= false;
END_ACTION

ACTION START_active:
xDone:=FALSE;
xTransCondition:= NOT xDone;
END_ACTION

TRANSITION TRANSITION:
xTransRelease AND xTransCondition
END_TRANSITION

END_FUNCTION_BLOCK

// ---- FBs/SUBFUNCTIONs/END_RUN_SEQ.TcPOU
FUNCTION_BLOCK END_RUN_SEQ
VAR_INPUT
	xJigEndDone:		BOOL;
END_VAR
VAR_IN_OUT
	xExecute:			BOOL;
	xDone:				BOOL;
END_VAR
VAR_OUTPUT
END_VAR
VAR
	tpReset:			TP;
	rtDone:				R_TRIG;
	rtExecute:			R_TRIG;
	ftTimePulse:		F_TRIG;
	tpTimePulse:		TP;
	lrTargetPos:		LREAL;
	
	xTransCondition:	BOOL;	
	xTransRelease:		BOOL;
	SFCInit:			BOOL;
	SFCReset:			BOOL;	
	SFCError:			BOOL;
END_VAR

rtDone(CLK:=xDone);
IF rtDone.Q THEN
	xTransRelease:=FALSE;	
	SFCReset:=TRUE;
	xExecute:=FALSE;
END_IF

rtExecute(CLK:=xExecute);
IF rtExecute.Q THEN
	xTransRelease:=TRUE;
END_IF

aSEQ_ACT();

tpReset(IN:=SFCError, PT:=T#250MS);
SFCReset:= tpReset.Q;

ACTION ACK_DONE_AXIS_active:
IF G_sAxisDone.X OR G_sAxisDone.Y OR G_sAxisDone.Z OR G_sAxisDone.c THEN
	G_sAckAxisDone.X:=TRUE;
	G_sAckAxisDone.Y:=TRUE;
	G_sAckAxisDone.Z:=TRUE;
	G_sAckAxisDone.C:=TRUE;
ELSE
	G_sAckAxisDone.X:=FALSE;
	G_sAckAxisDone.Y:=FALSE;
	G_sAckAxisDone.Z:=FALSE;
	G_sAckAxisDone.C:=FALSE;
END_IF

xTransCondition:= NOT G_sAckAxisDone.X AND NOT G_sAckAxisDone.Y AND NOT G_sAckAxisDone.Z AND NOT G_sAckAxisDone.C;
END_ACTION

ACTION aSEQ_ACT:
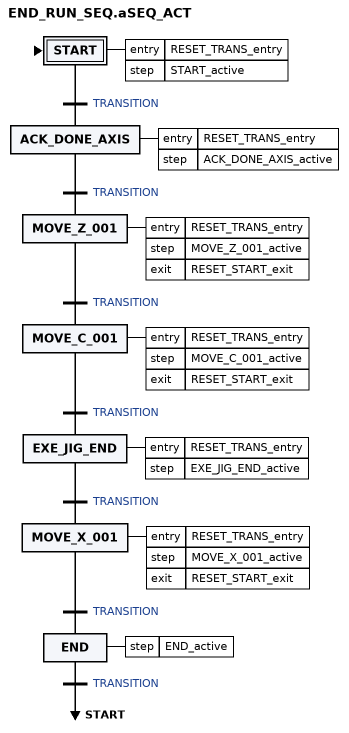
INITIAL_STEP START:
    RESET_TRANS_entry(P1);  // entry action
    START_active(N);  // step action
END_STEP
TRANSITION FROM START TO ACK_DONE_AXIS
    := TRANSITION;
END_TRANSITION
STEP ACK_DONE_AXIS:
    RESET_TRANS_entry(P1);  // entry action
    ACK_DONE_AXIS_active(N);  // step action
END_STEP
TRANSITION FROM ACK_DONE_AXIS TO MOVE_Z_001
    := TRANSITION;
END_TRANSITION
STEP MOVE_Z_001:
    RESET_TRANS_entry(P1);  // entry action
    MOVE_Z_001_active(N);  // step action
    RESET_START_exit(P0);  // exit action
END_STEP
TRANSITION FROM MOVE_Z_001 TO MOVE_C_001
    := TRANSITION;
END_TRANSITION
STEP MOVE_C_001:
    RESET_TRANS_entry(P1);  // entry action
    MOVE_C_001_active(N);  // step action
    RESET_START_exit(P0);  // exit action
END_STEP
TRANSITION FROM MOVE_C_001 TO EXE_JIG_END
    := TRANSITION;
END_TRANSITION
STEP EXE_JIG_END:
    RESET_TRANS_entry(P1);  // entry action
    EXE_JIG_END_active(N);  // step action
END_STEP
TRANSITION FROM EXE_JIG_END TO MOVE_X_001
    := TRANSITION;
END_TRANSITION
STEP MOVE_X_001:
    RESET_TRANS_entry(P1);  // entry action
    MOVE_X_001_active(N);  // step action
    RESET_START_exit(P0);  // exit action
END_STEP
TRANSITION FROM MOVE_X_001 TO END
    := TRANSITION;
END_TRANSITION
STEP END:
    END_active(N);  // step action
END_STEP
TRANSITION FROM END TO START
    := TRANSITION;
END_TRANSITION
END_ACTION

ACTION BLOW_DOWN_active:
tpTimePulse(IN:=NOT tpTimePulse.Q, PT:=T#3000MS);
ftTimePulse(CLK:=tpTimePulse.Q);
xTransCondition:= ftTimePulse.Q;
END_ACTION

ACTION END_active:
xDone:=TRUE;
xTransCondition:=xDone;
END_ACTION

ACTION EXE_JIG_END_active:
xTransCondition:=xJigEndDone;
END_ACTION

ACTION MOVE_C_001_active:
G_sControl.TargetPosition.C:= G_asIndividualAxisPositions[CE_AXIS_C].Positions[1].Target;
G_sStartToPos.C:= TRUE;

xTransCondition:= G_sAxisDone.C;
END_ACTION

ACTION MOVE_X_001_active:
G_sControl.TargetPosition.X:= G_asIndividualAxisPositions[CE_AXIS_X].Positions[1].Target;
G_sStartToPos.X:= TRUE;

xTransCondition:= G_sAxisDone.X;
END_ACTION

ACTION MOVE_Z_001_active:
G_sControl.TargetPosition.Z:= G_asIndividualAxisPositions[CE_AXIS_Z].Positions[1].Target;
G_sStartToPos.Z:= TRUE;

xTransCondition:= G_sAxisDone.Z;
END_ACTION

ACTION RESET_START_exit:
IF G_sAxisDone.X OR G_sAxisDone.Y OR G_sAxisDone.Z OR G_sAxisDone.c THEN
	G_sAckAxisDone.X:=TRUE;
	G_sAckAxisDone.Y:=TRUE;
	G_sAckAxisDone.Z:=TRUE;
	G_sAckAxisDone.C:=TRUE;
ELSE
	G_sAckAxisDone.X:=FALSE;
	G_sAckAxisDone.Y:=FALSE;
	G_sAckAxisDone.Z:=FALSE;
	G_sAckAxisDone.C:=FALSE;
	
	G_sStartToPos.X:=FALSE;
	G_sStartToPos.Y:=FALSE;
	G_sStartToPos.Z:=FALSE;
	G_sStartToPos.C:=FALSE;
END_IF
END_ACTION

ACTION RESET_TRANS_entry:
xTransCondition:= false;
END_ACTION

ACTION START_active:
xDone:=FALSE;
xTransCondition:= NOT xDone;
END_ACTION

TRANSITION TRANSITION:
xTransRelease AND xTransCondition
END_TRANSITION

END_FUNCTION_BLOCK

// ---- POUs/KERNEL POUs/OPERATIONs/SUBOPERATIONs/END_RUN.TcPOU
FUNCTION_BLOCK END_RUN
VAR_INPUT
END_VAR
VAR_OUTPUT
END_VAR
VAR
END_VAR

END_FUNCTION_BLOCK

// ---- POUs/KERNEL POUs/HMI_Controller.TcPOU
PROGRAM HMI_Controller
VAR
END_VAR

END_PROGRAM

// ---- FBs/DRIVEs/PNEU/PNEU_DRIVE.TcPOU
FUNCTION_BLOCK PNEU_DRIVE
VAR_INPUT
END_VAR
VAR_OUTPUT
END_VAR
VAR
END_VAR

END_FUNCTION_BLOCK

// ---- FBs/RECIPEs/CONVERTERs/ConvertCommandToString.TcPOU
FUNCTION_BLOCK ConvertCommandToString
VAR_INPUT
END_VAR
VAR_OUTPUT
END_VAR
VAR
END_VAR

END_FUNCTION_BLOCK

// ---- FBs/RECIPEs/CONVERTERs/CovertStringToCommand.TcPOU
FUNCTION_BLOCK CovertStringToCommand
VAR_INPUT
	
END_VAR
VAR_OUTPUT
END_VAR
VAR
END_VAR

END_FUNCTION_BLOCK

// ---- FBs/RECIPEs/FILEs/CreateRecipeFile.TcPOU
FUNCTION_BLOCK CreateRecipeFile
VAR_INPUT
END_VAR
VAR_OUTPUT
END_VAR
VAR
END_VAR

END_FUNCTION_BLOCK

// ---- FBs/RECIPEs/FILEs/ReadRecipeFromFile.TcPOU
FUNCTION_BLOCK ReadRecipeFromFile
VAR_INPUT
END_VAR
VAR_OUTPUT
END_VAR
VAR
END_VAR

END_FUNCTION_BLOCK

// ---- FBs/RECIPEs/FILEs/WriteRepcieToFile.TcPOU
FUNCTION_BLOCK WriteRepcieToFile
VAR_INPUT
END_VAR
VAR_OUTPUT
END_VAR
VAR
END_VAR

END_FUNCTION_BLOCK

// ---- FBs/SUBFUNCTIONs/PICKUP_SCREW_SEQ.TcPOU
FUNCTION_BLOCK PICKUP_SCREW_SEQ
VAR_IN_OUT
	xExecute:		BOOL;
END_VAR
VAR_OUTPUT
	xDone:			BOOL;
END_VAR
VAR
	tpReset:			TP;
	rtDone:				R_TRIG;
	rtExecute:			R_TRIG;
	ftTimePulse:		F_TRIG;
	tpTimePulse:		TP;
	lrTargetPos:		LREAL;
	xTransCondition:	BOOL;	
	xTransRelease:		BOOL;
	SFCInit:			BOOL;
	SFCReset:			BOOL;	
	SFCError:			BOOL;
END_VAR

rtDone(CLK:=xDone);
IF rtDone.Q THEN
	xTransRelease:=FALSE;	
	SFCReset:=TRUE;
END_IF

rtExecute(CLK:=xExecute);
IF rtExecute.Q THEN
	xTransRelease:=TRUE;
	SFCReset:=FALSE;
END_IF

IF xExecute THEN
	aSEQ_ACT();
END_IF

tpReset(IN:=SFCError, PT:=T#250MS);
SFCReset:= tpReset.Q;

ACTION ACK_DONE_AXIS_active:
IF G_sAxisDone.X OR G_sAxisDone.Y OR G_sAxisDone.Z OR G_sAxisDone.c THEN
	G_sAckAxisDone.X:=TRUE;
	G_sAckAxisDone.Y:=TRUE;
	G_sAckAxisDone.Z:=TRUE;
	G_sAckAxisDone.C:=TRUE;
ELSE
	G_sAckAxisDone.X:=FALSE;
	G_sAckAxisDone.Y:=FALSE;
	G_sAckAxisDone.Z:=FALSE;
	G_sAckAxisDone.C:=FALSE;
END_IF

xTransCondition:= NOT G_sAckAxisDone.X AND NOT G_sAckAxisDone.Y AND NOT G_sAckAxisDone.Z AND NOT G_sAckAxisDone.C;
END_ACTION

ACTION aSEQ_ACT:
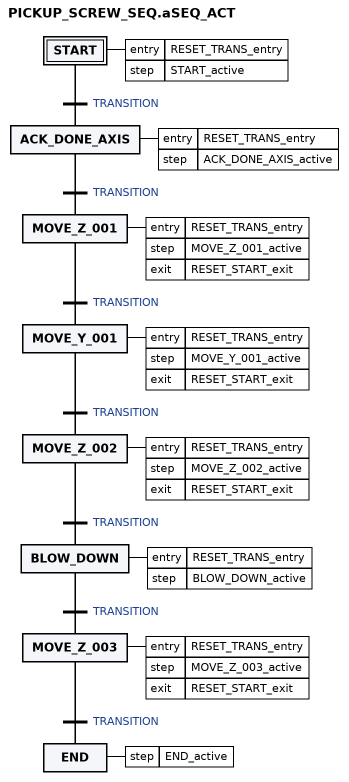
INITIAL_STEP START:
    RESET_TRANS_entry(P1);  // entry action
    START_active(N);  // step action
END_STEP
TRANSITION FROM START TO ACK_DONE_AXIS
    := TRANSITION;
END_TRANSITION
STEP ACK_DONE_AXIS:
    RESET_TRANS_entry(P1);  // entry action
    ACK_DONE_AXIS_active(N);  // step action
END_STEP
TRANSITION FROM ACK_DONE_AXIS TO MOVE_Z_001
    := TRANSITION;
END_TRANSITION
STEP MOVE_Z_001:
    RESET_TRANS_entry(P1);  // entry action
    MOVE_Z_001_active(N);  // step action
    RESET_START_exit(P0);  // exit action
END_STEP
TRANSITION FROM MOVE_Z_001 TO MOVE_Y_001
    := TRANSITION;
END_TRANSITION
STEP MOVE_Y_001:
    RESET_TRANS_entry(P1);  // entry action
    MOVE_Y_001_active(N);  // step action
    RESET_START_exit(P0);  // exit action
END_STEP
TRANSITION FROM MOVE_Y_001 TO MOVE_Z_002
    := TRANSITION;
END_TRANSITION
STEP MOVE_Z_002:
    RESET_TRANS_entry(P1);  // entry action
    MOVE_Z_002_active(N);  // step action
    RESET_START_exit(P0);  // exit action
END_STEP
TRANSITION FROM MOVE_Z_002 TO BLOW_DOWN
    := TRANSITION;
END_TRANSITION
STEP BLOW_DOWN:
    RESET_TRANS_entry(P1);  // entry action
    BLOW_DOWN_active(N);  // step action
END_STEP
TRANSITION FROM BLOW_DOWN TO MOVE_Z_003
    := TRANSITION;
END_TRANSITION
STEP MOVE_Z_003:
    RESET_TRANS_entry(P1);  // entry action
    MOVE_Z_003_active(N);  // step action
    RESET_START_exit(P0);  // exit action
END_STEP
TRANSITION FROM MOVE_Z_003 TO END
    := TRANSITION;
END_TRANSITION
STEP END:
    END_active(N);  // step action
END_STEP
END_ACTION

ACTION BLOW_DOWN_active:
tpTimePulse(IN:=NOT tpTimePulse.Q, PT:=T#3000MS);
ftTimePulse(CLK:=tpTimePulse.Q);
xTransCondition:= ftTimePulse.Q;
END_ACTION

ACTION END_active:
xDone:=TRUE;
xTransCondition:=FALSE;
END_ACTION

ACTION MOVE_Y_001_active:
G_sControl.TargetPosition.Y:= G_asIndividualAxisPositions[CE_AXIS_Y].Positions[1].Target;
G_sStartToPos.Y:= TRUE;

xTransCondition:= G_sAxisDone.Y;
END_ACTION

ACTION MOVE_Z_001_active:
G_sControl.TargetPosition.Z:= G_asIndividualAxisPositions[CE_AXIS_Z].Positions[1].Target;
G_sStartToPos.Z:= TRUE;

xTransCondition:= G_sAxisDone.Z;
END_ACTION

ACTION MOVE_Z_002_active:
G_sControl.TargetPosition.Z:= G_asIndividualAxisPositions[CE_AXIS_Z].Positions[2].Target;
G_sStartToPos.Z:= TRUE;

xTransCondition:= G_sAxisDone.Z;
END_ACTION

ACTION MOVE_Z_003_active:
G_sControl.TargetPosition.Z:= G_asIndividualAxisPositions[CE_AXIS_Z].Positions[1].Target;
G_sStartToPos.Z:= TRUE;

xTransCondition:= G_sAxisDone.Z;
END_ACTION

ACTION RESET_START_exit:
IF G_sAxisDone.X OR G_sAxisDone.Y OR G_sAxisDone.Z OR G_sAxisDone.c THEN
	G_sAckAxisDone.X:=TRUE;
	G_sAckAxisDone.Y:=TRUE;
	G_sAckAxisDone.Z:=TRUE;
	G_sAckAxisDone.C:=TRUE;
ELSE
	G_sAckAxisDone.X:=FALSE;
	G_sAckAxisDone.Y:=FALSE;
	G_sAckAxisDone.Z:=FALSE;
	G_sAckAxisDone.C:=FALSE;
	
	G_sStartToPos.X:=FALSE;
	G_sStartToPos.Y:=FALSE;
	G_sStartToPos.Z:=FALSE;
	G_sStartToPos.C:=FALSE;
END_IF
END_ACTION

ACTION RESET_TRANS_entry:
xTransCondition:= false;
END_ACTION

ACTION START_active:
xDone:=FALSE;
xTransCondition:= NOT xDone;
END_ACTION

TRANSITION TRANSITION:
xTransRelease AND xTransCondition
END_TRANSITION

END_FUNCTION_BLOCK

// ---- FBs/SUBFUNCTIONs/SELECT_ACTIVE_FEEDER_SEQ.TcPOU
FUNCTION_BLOCK SELECT_ACTIVE_FEEDER_SEQ
VAR_INPUT
	I_iActiveFeeder:				INT;
	I_axScrewFeederPosFeedback:		ARRAY [1..CE_SCREW_FEED_4] OF BOOL;
END_VAR
VAR_OUTPUT
	Q_xDone:						BOOL;	
	Q_axFeederValve:				ARRAY [1..CE_SCREW_FEED_4] OF BOOL;
END_VAR
VAR
END_VAR

CASE I_iActiveFeeder OF
	1:
		Q_axFeederValve[1]:=TRUE;
		Q_axFeederValve[2]:=FALSE;
	2:
		Q_axFeederValve[1]:=FALSE;
		Q_axFeederValve[2]:=TRUE;
	3:
		Q_axFeederValve[3]:=TRUE;
		Q_axFeederValve[4]:=FALSE;
	4:
		Q_axFeederValve[3]:=FALSE;
		Q_axFeederValve[4]:=TRUE;
END_CASE

IF Q_axFeederValve[I_iActiveFeeder]=I_axScrewFeederPosFeedback[I_iActiveFeeder] THEN
	Q_xDone:=TRUE;
ELSE
	Q_xDone:=FALSE;
END_IF

END_FUNCTION_BLOCK

// ---- POUs/JIG POUs/JIG TYPE POUs/JIG_EMPTY.TcPOU
PROGRAM JIG_EMPTY
VAR
END_VAR

END_PROGRAM

// ---- POUs/JIG POUs/JIG TYPE POUs/JIG_GRAB.TcPOU
PROGRAM JIG_GRAB
VAR
END_VAR

END_PROGRAM

// ---- POUs/JIG POUs/JIG TYPE POUs/JIG_PARTPRESENT.TcPOU
PROGRAM JIG_PARTPRESENT
VAR
END_VAR

END_PROGRAM

// ---- POUs/JIG POUs/JIG TYPE POUs/JIG_TAKER.TcPOU
PROGRAM JIG_TAKER
VAR
END_VAR

END_PROGRAM

// ---- POUs/JIG POUs/JIG001_VOLVOL125.TcPOU
PROGRAM JIG001_VOLVOL125
VAR
END_VAR

END_PROGRAM

// ---- POUs/JIG POUs/JIG002_MANSCANIA2016.TcPOU
PROGRAM JIG002_MANSCANIA2016
VAR
END_VAR

END_PROGRAM

// ---- POUs/JIG POUs/JIG003_NTG6.TcPOU
PROGRAM JIG003_NTG6
VAR
END_VAR

END_PROGRAM

// ---- POUs/JIG POUs/JIG004_BMW_RAM.TcPOU
PROGRAM JIG004_BMW_RAM
VAR
END_VAR

END_PROGRAM

// ---- POUs/JIG POUs/JIG005_BMW_MGU.TcPOU
PROGRAM JIG005_BMW_MGU
VAR
END_VAR

END_PROGRAM

// ---- POUs/KERNEL POUs/AST40_Controller.TcPOU
PROGRAM AST40_Controller
VAR
END_VAR

END_PROGRAM

// ---- POUs/KERNEL POUs/MES POUs/LOCAL_COM_Controller.TcPOU
PROGRAM LOCAL_COM_Controller
VAR
END_VAR

END_PROGRAM

// ---- POUs/KERNEL POUs/MES POUs/OPCUA_Controller.TcPOU
PROGRAM OPCUA_Controller
VAR
END_VAR

END_PROGRAM

// ---- POUs/KERNEL POUs/MES_Controller.TcPOU
PROGRAM MES_Controller
VAR
END_VAR

IF G_xComProtocol THEN
	OPCUA_Controller();
ELSE
	LOCAL_COM_Controller();
END_IF

END_PROGRAM

// ---- POUs/KERNEL POUs/OPERATIONs/AUTOMATIC_POSITION_TEST.TcPOU
FUNCTION_BLOCK AUTOMATIC_POSITION_TEST
VAR_INPUT
END_VAR
VAR_OUTPUT
END_VAR
VAR
END_VAR

ACTION ACT_SEQUENCE_CHAIN:
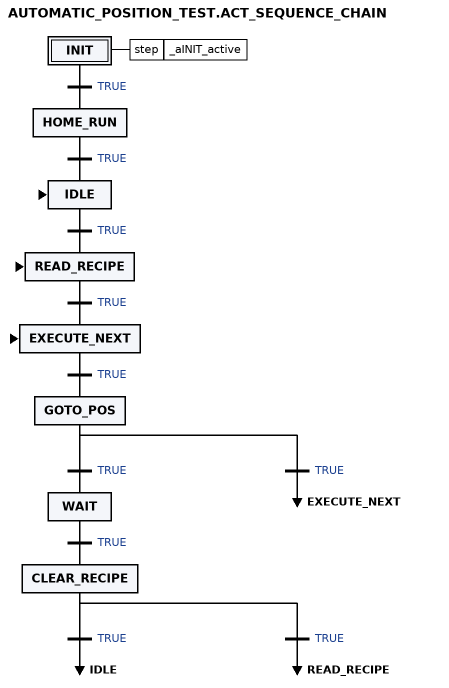
INITIAL_STEP INIT:
    _aINIT_active(N);  // step action
END_STEP
TRANSITION FROM INIT TO HOME_RUN
    := TRUE;
END_TRANSITION
STEP HOME_RUN:
END_STEP
TRANSITION FROM HOME_RUN TO IDLE
    := TRUE;
END_TRANSITION
STEP IDLE:
END_STEP
TRANSITION FROM IDLE TO READ_RECIPE
    := TRUE;
END_TRANSITION
STEP READ_RECIPE:
END_STEP
TRANSITION FROM READ_RECIPE TO EXECUTE_NEXT
    := TRUE;
END_TRANSITION
STEP EXECUTE_NEXT:
END_STEP
TRANSITION FROM EXECUTE_NEXT TO GOTO_POS
    := TRUE;
END_TRANSITION
STEP GOTO_POS:
END_STEP
TRANSITION FROM GOTO_POS TO WAIT
    := TRUE;
END_TRANSITION
TRANSITION FROM GOTO_POS TO EXECUTE_NEXT
    := TRUE;
END_TRANSITION
STEP WAIT:
END_STEP
TRANSITION FROM WAIT TO CLEAR_RECIPE
    := TRUE;
END_TRANSITION
STEP CLEAR_RECIPE:
END_STEP
TRANSITION FROM CLEAR_RECIPE TO IDLE
    := TRUE;
END_TRANSITION
TRANSITION FROM CLEAR_RECIPE TO READ_RECIPE
    := TRUE;
END_TRANSITION
// branch label Branch0_ACT_SEQUENCE_CHAIN
// branch label Branch1_ACT_SEQUENCE_CHAIN
END_ACTION

END_FUNCTION_BLOCK

// ---- POUs/KERNEL POUs/OPERATIONs/SUBOPERATIONs/HOME_RUN.TcPOU
FUNCTION_BLOCK HOME_RUN
VAR_INPUT
END_VAR
VAR_OUTPUT
END_VAR
VAR
END_VAR

END_FUNCTION_BLOCK

// ---- POUs/KERNEL POUs/OPERATIONs/AUTOMATIC_SCREWING.TcPOU
FUNCTION_BLOCK AUTOMATIC_SCREWING
VAR_INPUT
END_VAR
VAR_OUTPUT
END_VAR
VAR
END_VAR

ACTION ACT_SEQUENCE_CHAIN:
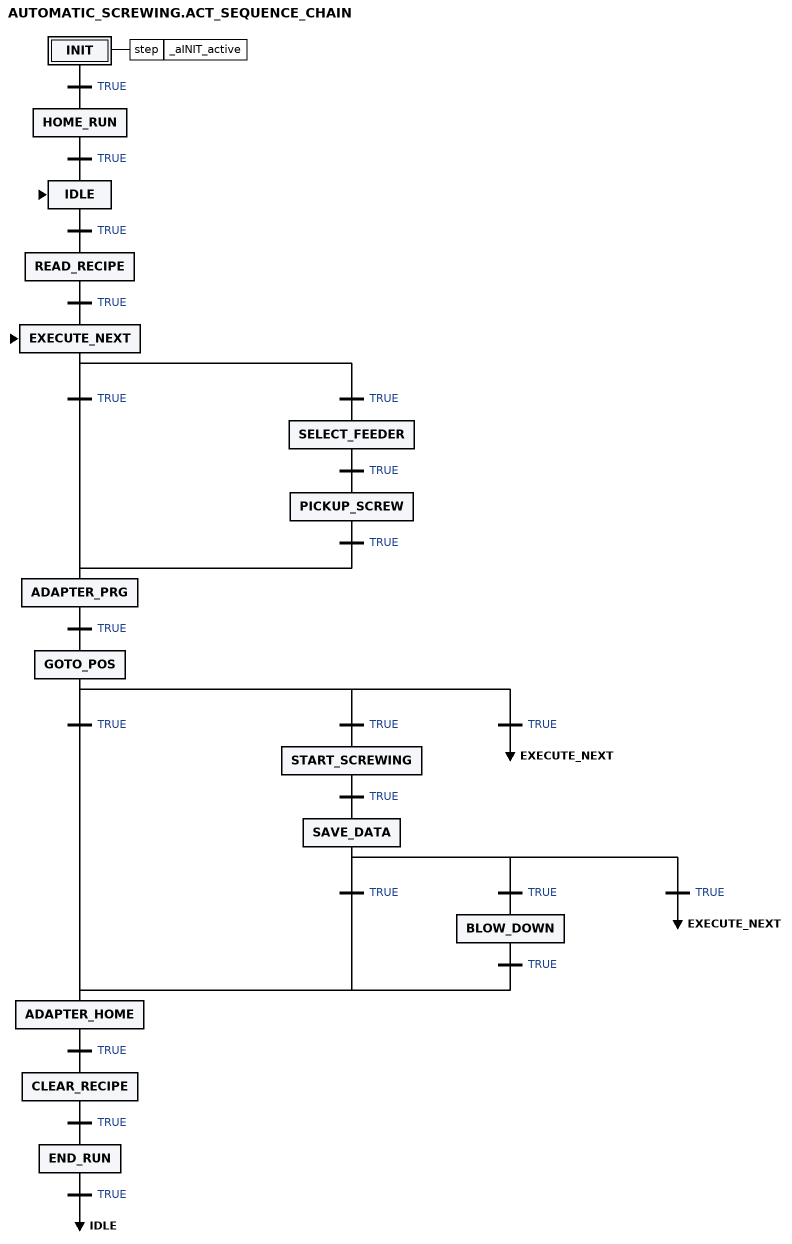
INITIAL_STEP INIT:
    _aINIT_active(N);  // step action
END_STEP
TRANSITION FROM INIT TO HOME_RUN
    := TRUE;
END_TRANSITION
STEP HOME_RUN:
END_STEP
TRANSITION FROM HOME_RUN TO IDLE
    := TRUE;
END_TRANSITION
STEP IDLE:
END_STEP
TRANSITION FROM IDLE TO READ_RECIPE
    := TRUE;
END_TRANSITION
STEP READ_RECIPE:
END_STEP
TRANSITION FROM READ_RECIPE TO EXECUTE_NEXT
    := TRUE;
END_TRANSITION
STEP EXECUTE_NEXT:
END_STEP
TRANSITION FROM EXECUTE_NEXT TO ADAPTER_PRG
    := TRUE;
END_TRANSITION
TRANSITION FROM EXECUTE_NEXT TO SELECT_FEEDER
    := TRUE;
END_TRANSITION
STEP SELECT_FEEDER:
END_STEP
TRANSITION FROM SELECT_FEEDER TO PICKUP_SCREW
    := TRUE;
END_TRANSITION
STEP PICKUP_SCREW:
END_STEP
TRANSITION FROM PICKUP_SCREW TO ADAPTER_PRG
    := TRUE;
END_TRANSITION
STEP ADAPTER_PRG:
END_STEP
TRANSITION FROM ADAPTER_PRG TO GOTO_POS
    := TRUE;
END_TRANSITION
STEP GOTO_POS:
END_STEP
TRANSITION FROM GOTO_POS TO ADAPTER_HOME
    := TRUE;
END_TRANSITION
TRANSITION FROM GOTO_POS TO START_SCREWING
    := TRUE;
END_TRANSITION
STEP START_SCREWING:
END_STEP
TRANSITION FROM START_SCREWING TO SAVE_DATA
    := TRUE;
END_TRANSITION
STEP SAVE_DATA:
END_STEP
TRANSITION FROM SAVE_DATA TO ADAPTER_HOME
    := TRUE;
END_TRANSITION
TRANSITION FROM SAVE_DATA TO BLOW_DOWN
    := TRUE;
END_TRANSITION
STEP BLOW_DOWN:
END_STEP
TRANSITION FROM BLOW_DOWN TO ADAPTER_HOME
    := TRUE;
END_TRANSITION
TRANSITION FROM SAVE_DATA TO EXECUTE_NEXT
    := TRUE;
END_TRANSITION
TRANSITION FROM GOTO_POS TO EXECUTE_NEXT
    := TRUE;
END_TRANSITION
STEP ADAPTER_HOME:
END_STEP
TRANSITION FROM ADAPTER_HOME TO CLEAR_RECIPE
    := TRUE;
END_TRANSITION
STEP CLEAR_RECIPE:
END_STEP
TRANSITION FROM CLEAR_RECIPE TO END_RUN
    := TRUE;
END_TRANSITION
STEP END_RUN:
END_STEP
TRANSITION FROM END_RUN TO IDLE
    := TRUE;
END_TRANSITION
// branch label Branch2_ACT_SEQUENCE_CHAIN
// branch label Branch3_ACT_SEQUENCE_CHAIN
// branch label Branch0_ACT_SEQUENCE_CHAIN
END_ACTION

END_FUNCTION_BLOCK

// ---- POUs/KERNEL POUs/OPERATIONs/SUBOPERATIONs/PICKUP_SCREW.TcPOU
FUNCTION_BLOCK PICKUP_SCREW
VAR_INPUT
END_VAR
VAR_OUTPUT
END_VAR
VAR
END_VAR

END_FUNCTION_BLOCK

// ---- POUs/KERNEL POUs/OPERATIONs/AUTOMATIC_SCREW_PICKUP_TEST.TcPOU
FUNCTION_BLOCK AUTOMATIC_SCREW_PICKUP_TEST
VAR_INPUT
END_VAR
VAR_OUTPUT
END_VAR
VAR
END_VAR

ACTION ACT_SEQUENCE_CHAIN:
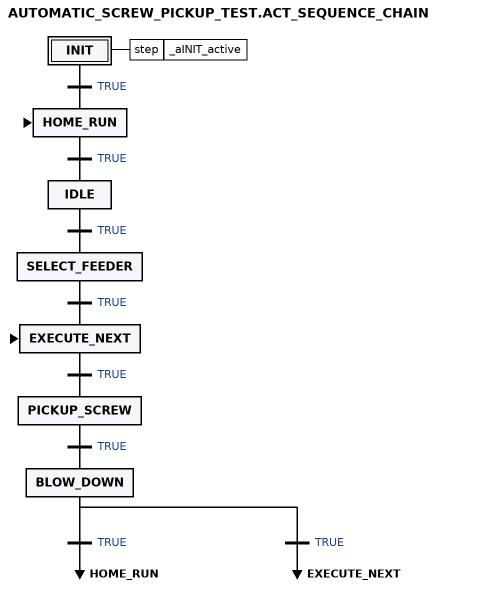
INITIAL_STEP INIT:
    _aINIT_active(N);  // step action
END_STEP
TRANSITION FROM INIT TO HOME_RUN
    := TRUE;
END_TRANSITION
STEP HOME_RUN:
END_STEP
TRANSITION FROM HOME_RUN TO IDLE
    := TRUE;
END_TRANSITION
STEP IDLE:
END_STEP
TRANSITION FROM IDLE TO SELECT_FEEDER
    := TRUE;
END_TRANSITION
STEP SELECT_FEEDER:
END_STEP
TRANSITION FROM SELECT_FEEDER TO EXECUTE_NEXT
    := TRUE;
END_TRANSITION
STEP EXECUTE_NEXT:
END_STEP
TRANSITION FROM EXECUTE_NEXT TO PICKUP_SCREW
    := TRUE;
END_TRANSITION
STEP PICKUP_SCREW:
END_STEP
TRANSITION FROM PICKUP_SCREW TO BLOW_DOWN
    := TRUE;
END_TRANSITION
STEP BLOW_DOWN:
END_STEP
TRANSITION FROM BLOW_DOWN TO HOME_RUN
    := TRUE;
END_TRANSITION
TRANSITION FROM BLOW_DOWN TO EXECUTE_NEXT
    := TRUE;
END_TRANSITION
// branch label Branch0_ACT_SEQUENCE_CHAIN
END_ACTION

END_FUNCTION_BLOCK

// ---- POUs/KERNEL POUs/OPERATIONs/SUBOPERATIONs/DROP_SCREW.TcPOU
FUNCTION_BLOCK DROP_SCREW
VAR_INPUT
END_VAR
VAR_OUTPUT
END_VAR
VAR
END_VAR

END_FUNCTION_BLOCK

// ---- POUs/KERNEL POUs/OPERATIONs/SUBOPERATIONs/POSITION_RUN.TcPOU
FUNCTION_BLOCK POSITION_RUN
VAR_INPUT
END_VAR
VAR_OUTPUT
END_VAR
VAR
END_VAR

END_FUNCTION_BLOCK

// ---- POUs/KERNEL POUs/RECIPE_Controller.TcPOU
PROGRAM RECIPE_Controller
VAR	
	xExecuteNextLine:		BOOL;
	xDoneActualLine:		BOOL;
	nCommandID:				INT;
	nAdapterParameter:		INT;
	nTargetFeeder:			INT;
	nScrewingProgram:		INT;
	sGoToTraget:			tsCoordinateBool;
	sTargetCoordinate:		tsCoordinate;	
END_VAR

(*
	Recipe read from file, write to file, and create new
*)

END_PROGRAM

// ---- POUs/MAIN POUs/INDEP.TcPOU
PROGRAM INDEP
VAR
END_VAR

END_PROGRAM

// ---- POUs/MAIN POUs/JIG.TcPOU
PROGRAM JIG
VAR
END_VAR

END_PROGRAM
